   1:  PR[91,2] = PR[90,2] + -28.549;
   1:L PR[91] R[100]mm/sec CNT100;
   1:  PR[91,1] = PR[90,1] + 41.610;
   1:  PR[91,2] = PR[90,2] + -32.305;
   1:L PR[91] R[100]mm/sec CNT100;
   1:  PR[91,1] = PR[90,1] + 47.267;
   1:  PR[91,2] = PR[90,2] + -33.357;
   1:L PR[91] R[100]mm/sec CNT100;
   1:  PR[91,1] = PR[90,1] + 47.490;
   1:  PR[91,2] = PR[90,2] + -33.379;
   1:L PR[91] R[100]mm/sec CNT100;
   1:  PR[91,1] = PR[90,1] + 53.158;
   1:  PR[91,2] = PR[90,2] + -33.726;
   1:L PR[91] R[100]mm/sec CNT100;
   1:  PR[91,1] = PR[90,1] + 53.368;
   1:  PR[91,2] = PR[90,2] + -33.724;
   1:L PR[91] R[100]mm/sec CNT100;
   1:  PR[91,1] = PR[90,1] + 59.077;
   1:  PR[91,2] = PR[90,2] + -33.374;
   1:L PR[91] R[100]mm/sec CNT100;
   1:  PR[91,1] = PR[90,1] + 59.253;
   1:  PR[91,2] = PR[90,2] + -33.352;
   1:L PR[91] R[100]mm/sec CNT100;
   1:  PR[91,1] = PR[90,1] + 64.813;
   1:  PR[91,2] = PR[90,2] + -32.326;
   1:L PR[91] R[100]mm/sec CNT100;
   1:  PR[91,1] = PR[90,1] + 64.906;
   1:  PR[91,2] = PR[90,2] + -32.304;
   1:L PR[91] R[100]mm/sec CNT100;
   1:  PR[91,1] = PR[90,1] + 64.993;
   1:  PR[91,2] = PR[90,2] + -32.271;
   1:L PR[91] R[100]mm/sec CNT100;
   1:  PR[91,1] = PR[90,1] + 75.220;
   1:  PR[91,2] = PR[90,2] + -28.355;
   1:L PR[91] R[100]mm/sec CNT100;
   1:  PR[91,1] = PR[90,1] + 83.384;
   1:  PR[91,2] = PR[90,2] + -22.557;
   1:L PR[91] R[100]mm/sec CNT100;
   1:  PR[91,1] = PR[90,1] + 89.083;
   1:  PR[91,2] = PR[90,2] + -15.676;
   1:L PR[91] R[100]mm/sec CNT100;
   1:  PR[91,1] = PR[90,1] + 92.383;
   1:  PR[91,2] = PR[90,2] + -8.281;
   1:L PR[91] R[100]mm/sec CNT100;
   1:  PR[91,1] = PR[90,1] + 93.446;
   1:  PR[91,2] = PR[90,2] + -0.729;
   1:L PR[91] R[100]mm/sec CNT100;
   1:  PR[91,1] = PR[90,1] + 92.381;
   1:  PR[91,2] = PR[90,2] + 6.834;
   1:L PR[91] R[100]mm/sec CNT100;
   1:  PR[91,1] = PR[90,1] + 89.082;
   1:  PR[91,2] = PR[90,2] + 14.219;
   1:L PR[91] R[100]mm/sec CNT100;
   1:  PR[91,1] = PR[90,1] + 83.380;
   1:  PR[91,2] = PR[90,2] + 21.102;
   1:L PR[91] R[100]mm/sec CNT100;
   1:  PR[91,1] = PR[90,1] + 75.215;
   1:  PR[91,2] = PR[90,2] + 26.899;
   1:L PR[91] R[100]mm/sec CNT100;
   1:  PR[91,1] = PR[90,1] + 64.892;
   1:  PR[91,2] = PR[90,2] + 30.848;
   1:L PR[91] R[100]mm/sec CNT100;
   1:  PR[91,1] = PR[90,1] + 64.807;
   1:  PR[91,2] = PR[90,2] + 30.868;
   1:L PR[91] R[100]mm/sec CNT100;
   1:  PR[91,1] = PR[90,1] + 59.247;
   1:  PR[91,2] = PR[90,2] + 31.894;
   1:L PR[91] R[100]mm/sec CNT100;
   1:  PR[91,1] = PR[90,1] + 59.072;
   1:  PR[91,2] = PR[90,2] + 31.916;
   1:L PR[91] R[100]mm/sec CNT100;
   1:  PR[91,1] = PR[90,1] + 53.363;
   1:  PR[91,2] = PR[90,2] + 32.265;
   1:L PR[91] R[100]mm/sec CNT100;
   1:  PR[91,1] = PR[90,1] + 53.153;
   1:  PR[91,2] = PR[90,2] + 32.267;
   1:L PR[91] R[100]mm/sec CNT100;
   1:  PR[91,1] = PR[90,1] + 47.485;
   1:  PR[91,2] = PR[90,2] + 31.919;
   1:L PR[91] R[100]mm/sec CNT100;
   1:  PR[91,1] = PR[90,1] + 47.260;
   1:  PR[91,2] = PR[90,2] + 31.897;
   1:L PR[91] R[100]mm/sec CNT100;
   1:  PR[91,1] = PR[90,1] + 41.822;
   1:  PR[91,2] = PR[90,2] + 30.893;
   1:L PR[91] R[100]mm/sec CNT100;
   1:  PR[91,1] = PR[90,1] + 41.569;
   1:  PR[91,2] = PR[90,2] + 30.841;
   1:L PR[91] R[100]mm/sec CNT100;
   1:  PR[91,1] = PR[90,1] + 41.262;
   1:  PR[91,2] = PR[90,2] + 30.742;
   1:L PR[91] R[100]mm/sec CNT100;
   1:  PR[91,1] = PR[90,1] + 40.649;
   1:  PR[91,2] = PR[90,2] + 30.481;
   1:L PR[91] R[100]mm/sec CNT100;
   1:  PR[91,1] = PR[90,1] + 31.250;
   1:  PR[91,2] = PR[90,2] + 26.882;
   1:L PR[91] R[100]mm/sec CNT100;
   1:  PR[91,1] = PR[90,1] + 30.868;
   1:  PR[91,2] = PR[90,2] + 26.654;
   1:L PR[91] R[100]mm/sec CNT100;
   1:  PR[91,1] = PR[90,1] + 30.063;
   1:  PR[91,2] = PR[90,2] + 26.056;
   1:L PR[91] R[100]mm/sec CNT100;
   1:  PR[91,1] = PR[90,1] + 23.191;
   1:  PR[91,2] = PR[90,2] + 21.173;
   1:L PR[91] R[100]mm/sec CNT100;
   1:  PR[91,1] = PR[90,1] + 22.612;
   1:  PR[91,2] = PR[90,2] + 20.595;
   1:L PR[91] R[100]mm/sec CNT100;
   1:  PR[91,1] = PR[90,1] + 21.528;
   1:  PR[91,2] = PR[90,2] + 19.243;
   1:L PR[91] R[100]mm/sec CNT100;
   1:  PR[91,1] = PR[90,1] + 17.552;
   1:  PR[91,2] = PR[90,2] + 14.442;
   1:L PR[91] R[100]mm/sec CNT100;
   1:  PR[91,1] = PR[90,1] + 16.754;
   1:  PR[91,2] = PR[90,2] + 13.031;
   1:L PR[91] R[100]mm/sec CNT100;
   1:  PR[91,1] = PR[90,1] + 15.495;
   1:  PR[91,2] = PR[90,2] + 10.029;
   1:L PR[91] R[100]mm/sec CNT100;
   1:  PR[91,1] = PR[90,1] + 14.201;
   1:  PR[91,2] = PR[90,2] + 7.134;
   1:L PR[91] R[100]mm/sec CNT100;
   1:  PR[91,1] = PR[90,1] + 13.515;
   1:  PR[91,2] = PR[90,2] + 4.130;
   1:L PR[91] R[100]mm/sec CNT100 TB   .50sec,CALL END_PUD;
   1:  DO[117:Laser Start]=OFF;
   1:  PR[92] = PR[91];
   1:  PR[92,3] = PR[92,3] + 50;
   1:J PR[92] 10% FINE;
   1:  WAIT   5.00(sec);
   1:  DO[119:Gas]=OFF;
   1:  CALL HOME_ALL;
/POS
/END
